(* Logix 5000 project; controller Safety vendor 1 type 14 code 148 rev 32.11; software revision 32.03; part 11 of 17 *)
(* tags used below, declared in another part *)
   ExBridle_DrvsOff : BOOL;   // Exit Bridle Drives OFF ( 1= OFF)
   ExBridle_SafeOffEn : BOOL;   // Exit Bridle Safe-Off Enable ( 1= Enable )
   ExBridle_SafeOffFltRst : BOOL;   // Exit Bridle Safe-Off Fault Reset ( 1= Reset Cmd )
   Line_TotalMode : BOOL;   // Line TOTAL Mode ( 1= Total Mode) (0 = Coil to Coil)
   LineSts : UDT_SysStatus;
   PW_DrvsOff : BOOL;   // Paper Winder Drives OFF ( 1= OFF)
   PW_SafeTrqEn : BOOL;   // Paper Winder Safe-Trq Off Enable ( 1= Enable )
   Rew_DrvsOff : BOOL;   // Rewind Drives OFF ( 1= OFF)
   REW_SafeOffEn : BOOL;   // Rewind Safe-Off Enable ( 1= Enable )
   REW_SafeOffFltRst : BOOL;   // Rewind Safe-Off Fault Reset ( 1= Reset Cmd )
   SafeOff_y172CR460 : CONFIGURABLE_ROUT;   // Shear Die Main Contactor Relay
   SafeOff_y172CR460_Flt : ALIAS FOR Flt_SafeOff[0].0;   // Shear Die Main Contactor Relay Fault ( 1= Fault)
   SafeOff_y172CR510 : CONFIGURABLE_ROUT;   // Shear Die Drive Enable Relay
   SafeOff_y172CR510_Flt : ALIAS FOR Flt_SafeOff[0].1;   // Shear Die Drive Enable Relay Fault ( 1= Fault)
   SafeOff_y614CR040 : CONFIGURABLE_ROUT;   // #1 Exit Bridle Roll 6 Main Contactor Relay
   SafeOff_y614CR040_Flt : ALIAS FOR Flt_SafeOff[0].10;   // #1 Exit Bridle Roll 6 Main Contactor Relay Fault ( 1= Fault)
   SafeOff_y614CR090 : CONFIGURABLE_ROUT;   // #1 Exit Bridle Roll 6 Drive Enable Relay
   SafeOff_y614CR090_Flt : ALIAS FOR Flt_SafeOff[0].11;   // #1 Exit Bridle Roll 6 Drive Enable Relay Fault ( 1= Fault)
   SafeOff_y614CR130 : CONFIGURABLE_ROUT;   // #2 Exit Bridle Roll 7 Main Contactor Relay
   SafeOff_y614CR130_Flt : ALIAS FOR Flt_SafeOff[0].12;   // #2 Exit Bridle Roll 7 Main Contactor Relay Fault ( 1= Fault)
   SafeOff_y614CR170 : CONFIGURABLE_ROUT;   // #2 Exit Bridle Roll 7 Drive Enable Relay
   SafeOff_y614CR170_Flt : ALIAS FOR Flt_SafeOff[0].13;   // #2 Exit Bridle Roll 7 Drive Enable Relay Fault ( 1= Fault)
   SafeOff_y614CR210 : CONFIGURABLE_ROUT;   // Rewind Main Contactor Relay
   SafeOff_y614CR210_Flt : ALIAS FOR Flt_SafeOff[0].14;   // Rewind Main Contactor Relay Fault ( 1= Fault)
   SafeOff_y614CR250 : CONFIGURABLE_ROUT;   // Rewind Drive Enable Relay
   SafeOff_y614CR250_Flt : ALIAS FOR Flt_SafeOff[0].15;   // Rewind Drive Enable Relay Fault ( 1= Fault)
   SC_DrvsOff : BOOL;   // Scrap Chop Conveyor Drives OFF ( 1= OFF)
   SC_SafeTrqEn : BOOL;   // Scrap Chopper Safe-Trq Off Enable ( 1= Enable )
   SGWA_DrvsOff : BOOL;   // Side Guide Width Adjust Drives OFF ( 1= OFF)
   SGWA_SafeTrqEn : BOOL;   // Side Guide Width Adjust Safe-Trq Off Enable ( 1= Enable )
   ShearSts : UDT_ShearStatus;
   SrDie_DrvsOff : BOOL;   // Shear Die Drives OFF ( 1= OFF)
   SrDie_SafeOffEn : BOOL;   // Shear Die Safe-Off Enable ( 1= Enable )
   SrDie_SafeOffFltRst : BOOL;   // Shear Die Safe-Off Fault Reset ( 1= Reset Cmd )
   TK_DrvsOff : BOOL;   // Trimmer Knives/ Width Adjust Drives OFF ( 1= OFF)
   TK_SafeTrqEn : BOOL;   // Trimmer Knife Safe-Trq Off Enable ( 1= Enable )
   UnPR_DrvsOff : BOOL;   // Unwind Pinch Roll Drives OFF ( 1= OFF)
   UnPR_SafeTrqEn : BOOL;   // Unwind Pinch Roll Safe-Trq Off Enable ( 1= Enable )
   WTPR_DrvsOff : BOOL;   // Wash Tank Pinch Rolls (1-4) Drives OFF ( 1= OFF)
   WTPR_SafeTrqEn : BOOL;   // Wash Tank Pinch Rolls (1-4) Safe-Trq Off Enable ( 1= Enable )
   x172CR460 : ALIAS FOR SDPLC:1:I.Pt00Data;   // Shear Die Drive Main Contactor Safety Relay Input
   x172CR510 : ALIAS FOR SDPLC:1:I.Pt01Data;   // Shear Die Drive Enable Safety Relay Input
   x614CR040 : ALIAS FOR CHPLC:2:I.Pt00Data;   // #1 Exit Bridle Roll 6 Main Contactor Safety Relay
   x614CR090 : ALIAS FOR CHPLC:2:I.Pt01Data;   // #1 Exit Bridle Roll 6 Drive Enable Safety Relay
   x614CR130 : ALIAS FOR CHPLC:2:I.Pt02Data;   // #2 Exit Bridle Roll 7 Main Contactor Safety Relay
   x614CR170 : ALIAS FOR CHPLC:2:I.Pt03Data;   // #2 Exit Bridle Roll 7 Drive Enable Safety Relay
   x614CR210 : ALIAS FOR CHPLC:2:I.Pt04Data;   // Rewind Main Contactor Safety Relay
   x614CR250 : ALIAS FOR CHPLC:2:I.Pt05Data;   // Rewind Drive Enable Safety Relay
   x759MTR080SE : ALIAS FOR MCC3:4:O.Pt02Data;   // Scrap Choppers Width Adjust Safety Enable
   x759MTR080SP : ALIAS FOR MCC3:4:O.Pt01Data;   // Scrap Choppers Width Adjust Safety Power
   y172CR460 : ALIAS FOR SDPLC:2:O.Pt00Data;   // Shear Die Drive Main Contactor Safety Relay Output
   y172CR510 : ALIAS FOR SDPLC:2:O.Pt01Data;   // Shear Die Drive Enable Safety Relay Output
   y614CR040 : ALIAS FOR CHPLC:5:O.Pt00Data;   // #1 Exit Bridle Roll 6 Main Contactor Safety Relay
   y614CR090 : ALIAS FOR CHPLC:5:O.Pt01Data;   // #1 Exit Bridle Roll 6 Drive Enable Safety Relay
   y614CR130 : ALIAS FOR CHPLC:5:O.Pt02Data;   // #2 Exit Bridle Roll 7 Main Contactor Safety Relay
   y614CR170 : ALIAS FOR CHPLC:5:O.Pt03Data;   // #2 Exit Bridle Roll 7 Drive Enable Safety Relay
   y614CR210 : ALIAS FOR CHPLC:5:O.Pt04Data;   // Rewind Main Contactor Safety Relay
   y614CR250 : ALIAS FOR CHPLC:5:O.Pt05Data;   // Rewind Drive Enable Safety Relay
   y725MTR080SE : ALIAS FOR MCC2:1:O.Pt01Data;   // Unwind Pinch Roll Safety Enable
   y725MTR080SP : ALIAS FOR MCC2:1:O.Pt00Data;   // Unwind Pinch Roll Safety Power
   y727MTR080SE : ALIAS FOR MCC2:1:O.Pt05Data;   // Paper Winder Safety Enable
   y727MTR080SP : ALIAS FOR MCC2:1:O.Pt04Data;   // Paper Winder Safety Power
   y729MTR080SE : ALIAS FOR MCC2:1:O.Pt03Data;   // Washtank Pinch Roll 4 Safety Enable
   y729MTR080SP : ALIAS FOR MCC2:1:O.Pt02Data;   // Washtank Pinch Roll 4 Safety Power
   y731MTR080SE : ALIAS FOR MCC2:1:O.Pt07Data;   // Washtank Pinch Roll 1 Safety Enable
   y731MTR080SP : ALIAS FOR MCC2:1:O.Pt06Data;   // Washtank Pinch Roll 1 Safety Power
   y733MTR080SE : ALIAS FOR MCC2:2:O.Pt01Data;   // Washtank Pinch Roll 2 Safety Enable
   y733MTR080SP : ALIAS FOR MCC2:2:O.Pt00Data;   // Washtank Pinch Roll 2 Safety Power
   y735MTR080SE : ALIAS FOR MCC2:2:O.Pt03Data;   // Washtank Pinch Roll 3 Safety Enable
   y735MTR080SP : ALIAS FOR MCC2:2:O.Pt02Data;   // Washtank Pinch Roll 3 Safety Power
   y751MTR080SE : ALIAS FOR MCC3:3:O.Pt04Data;   // Trimmer Knives Safety Enable
   y751MTR080SP : ALIAS FOR MCC3:3:O.Pt03Data;   // Trimmer Knives Safety Power
   y754MTR080SE : ALIAS FOR MCC3:3:O.Pt06Data;   // Side Guide Width Adjust Safety Enable
   y754MTR080SP : ALIAS FOR MCC3:3:O.Pt05Data;   // Side Guide Width Adjust Safety Power
   y755MTR080SE : ALIAS FOR MCC3:4:O.Pt00Data;   // Trimmer Knives Width Adjust Safety Enable
   y755MTR080SP : ALIAS FOR MCC3:3:O.Pt07Data;   // Trimmer Knives Width Adjust Safety Power
   y762MTR080SE : ALIAS FOR MCC3:4:O.Pt04Data;   // Scrap Choppers Safety Enable
   y762MTR080SP : ALIAS FOR MCC3:4:O.Pt03Data;   // Scrap Choppers Safety Power
(* SafeOff, continued *)

ROUTINE A03_ExitBridle_CR   (* ladder *)
// Exit Bridle
// Main Contactor and Drive Enable
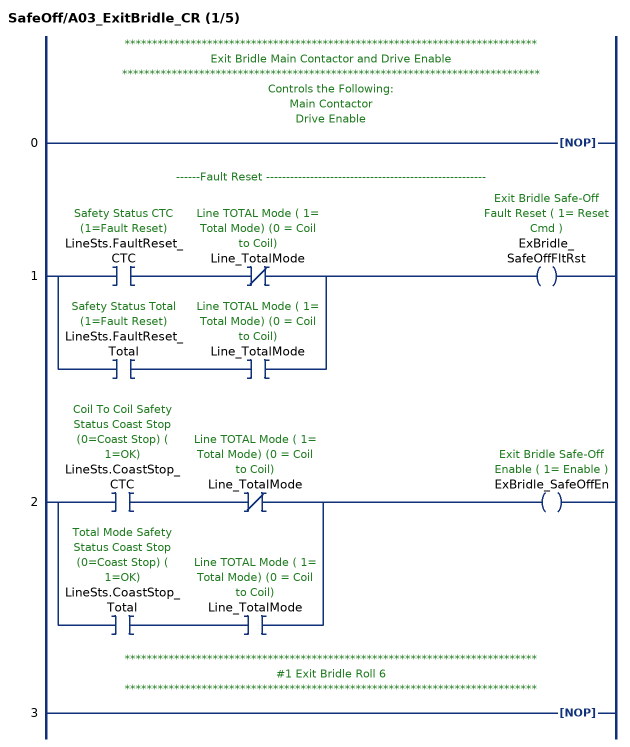
   // ***************************************************************************
   // Exit Bridle Main Contactor and Drive Enable
   // ****************************************************************************
   // Controls the Following:
   // Main Contactor
   // Drive Enable
   0: NOP();
   // ------Fault Reset -------------------------------------------------------
   1: [XIC(LineSts.FaultReset_CTC) XIO(Line_TotalMode) ,XIC(LineSts.FaultReset_Total) XIC(Line_TotalMode) ]OTE(ExBridle_SafeOffFltRst);
   2: [XIC(LineSts.CoastStop_CTC) XIO(Line_TotalMode) ,XIC(LineSts.CoastStop_Total) XIC(Line_TotalMode) ]OTE(ExBridle_SafeOffEn);
   // ***************************************************************************
   // #1 Exit Bridle Roll 6
   // ***************************************************************************
   3: NOP();
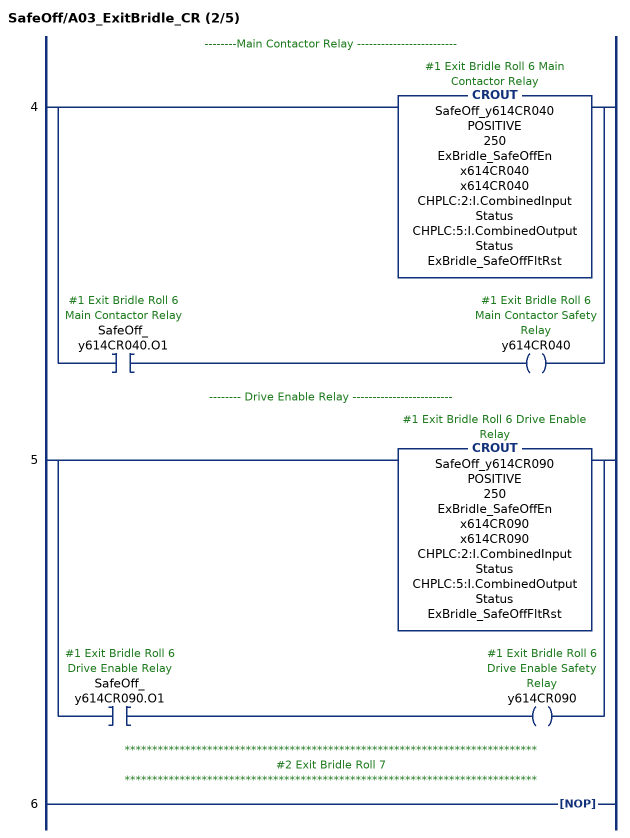
   // --------Main Contactor Relay -------------------------
   4: [CROUT(SafeOff_y614CR040,POSITIVE,250,ExBridle_SafeOffEn,x614CR040,x614CR040,CHPLC:2:I.CombinedInputStatus,CHPLC:5:I.CombinedOutputStatus,ExBridle_SafeOffFltRst) ,XIC(SafeOff_y614CR040.O1) OTE(y614CR040) ];
   // -------- Drive Enable Relay -------------------------
   5: [CROUT(SafeOff_y614CR090,POSITIVE,250,ExBridle_SafeOffEn,x614CR090,x614CR090,CHPLC:2:I.CombinedInputStatus,CHPLC:5:I.CombinedOutputStatus,ExBridle_SafeOffFltRst) ,XIC(SafeOff_y614CR090.O1) OTE(y614CR090) ];
   // ***************************************************************************
   // #2 Exit Bridle Roll 7
   // ***************************************************************************
   6: NOP();
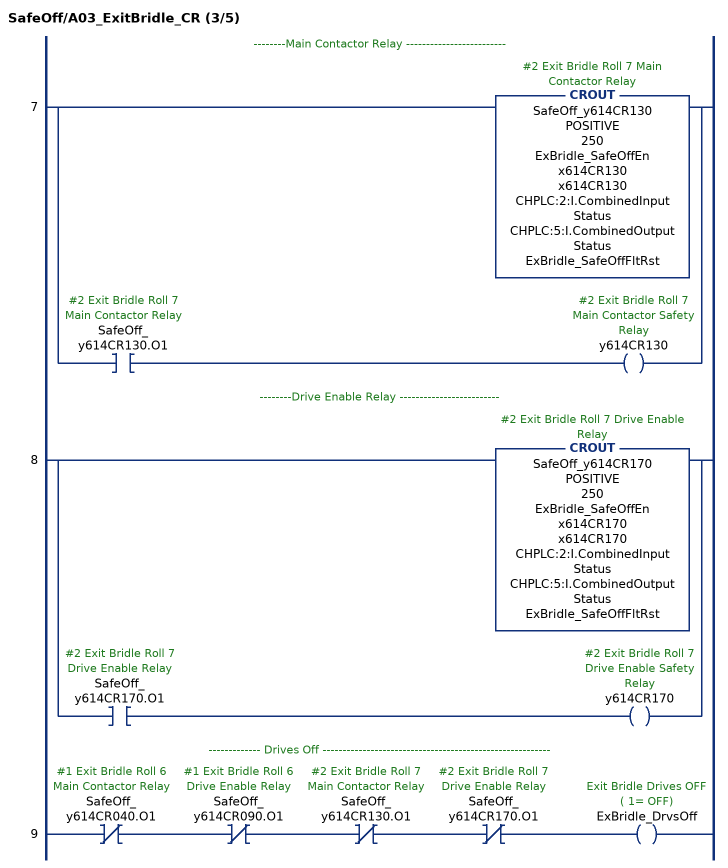
   // --------Main Contactor Relay -------------------------
   7: [CROUT(SafeOff_y614CR130,POSITIVE,250,ExBridle_SafeOffEn,x614CR130,x614CR130,CHPLC:2:I.CombinedInputStatus,CHPLC:5:I.CombinedOutputStatus,ExBridle_SafeOffFltRst) ,XIC(SafeOff_y614CR130.O1) OTE(y614CR130) ];
   // --------Drive Enable Relay -------------------------
   8: [CROUT(SafeOff_y614CR170,POSITIVE,250,ExBridle_SafeOffEn,x614CR170,x614CR170,CHPLC:2:I.CombinedInputStatus,CHPLC:5:I.CombinedOutputStatus,ExBridle_SafeOffFltRst) ,XIC(SafeOff_y614CR170.O1) OTE(y614CR170) ];
   // ------------- Drives Off ---------------------------------------------------------
   9: XIO(SafeOff_y614CR040.O1)XIO(SafeOff_y614CR090.O1)XIO(SafeOff_y614CR130.O1)XIO(SafeOff_y614CR170.O1)OTE(ExBridle_DrvsOff);
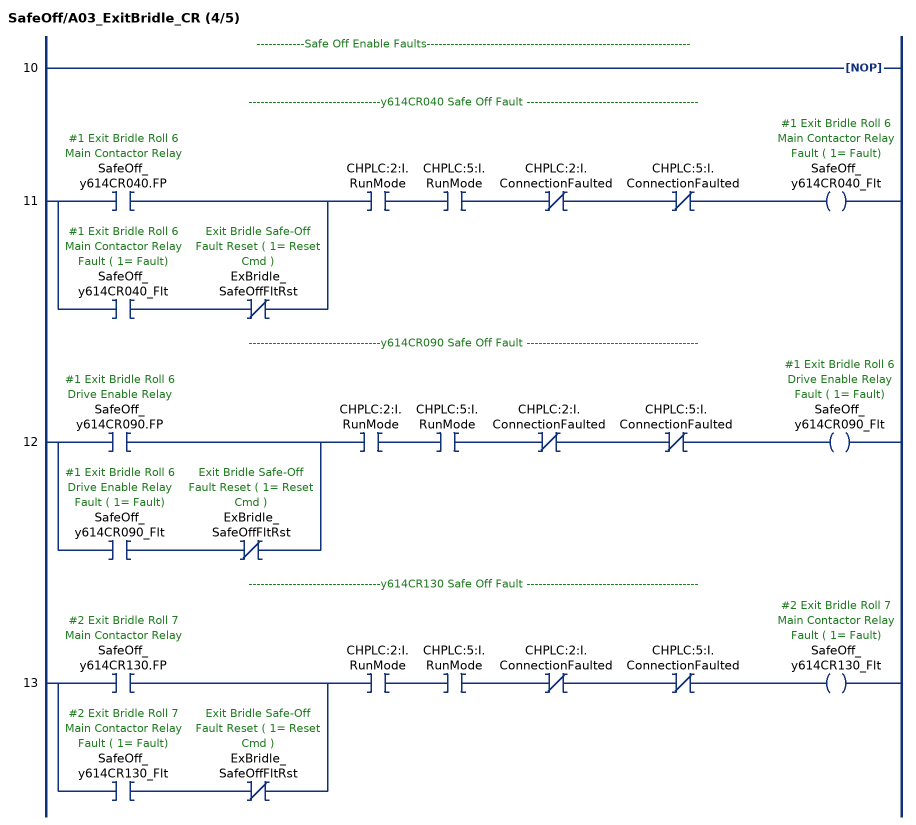
   // ------------Safe Off Enable Faults------------------------------------------------------------------
   10: NOP();
   // ---------------------------------y614CR040 Safe Off Fault -------------------------------------------
   11: [XIC(SafeOff_y614CR040.FP) ,XIC(SafeOff_y614CR040_Flt) XIO(ExBridle_SafeOffFltRst) ]XIC(CHPLC:2:I.RunMode)XIC(CHPLC:5:I.RunMode)XIO(CHPLC:2:I.ConnectionFaulted)XIO(CHPLC:5:I.ConnectionFaulted)OTE(SafeOff_y614CR040_Flt);
   // ---------------------------------y614CR090 Safe Off Fault -------------------------------------------
   12: [XIC(SafeOff_y614CR090.FP) ,XIC(SafeOff_y614CR090_Flt) XIO(ExBridle_SafeOffFltRst) ]XIC(CHPLC:2:I.RunMode)XIC(CHPLC:5:I.RunMode)XIO(CHPLC:2:I.ConnectionFaulted)XIO(CHPLC:5:I.ConnectionFaulted)OTE(SafeOff_y614CR090_Flt);
   // ---------------------------------y614CR130 Safe Off Fault -------------------------------------------
   13: [XIC(SafeOff_y614CR130.FP) ,XIC(SafeOff_y614CR130_Flt) XIO(ExBridle_SafeOffFltRst) ]XIC(CHPLC:2:I.RunMode)XIC(CHPLC:5:I.RunMode)XIO(CHPLC:2:I.ConnectionFaulted)XIO(CHPLC:5:I.ConnectionFaulted)OTE(SafeOff_y614CR130_Flt);
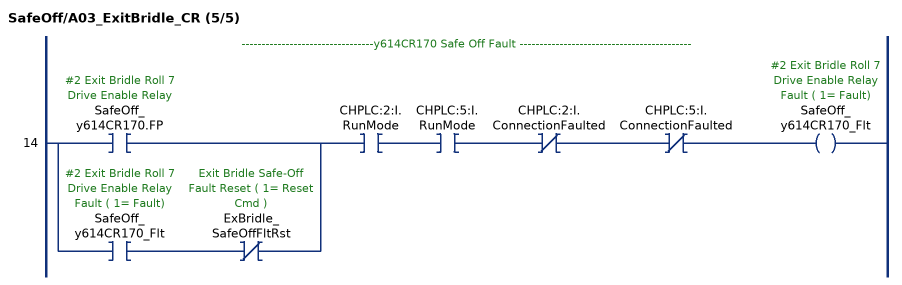
   // ---------------------------------y614CR170 Safe Off Fault -------------------------------------------
   14: [XIC(SafeOff_y614CR170.FP) ,XIC(SafeOff_y614CR170_Flt) XIO(ExBridle_SafeOffFltRst) ]XIC(CHPLC:2:I.RunMode)XIC(CHPLC:5:I.RunMode)XIO(CHPLC:2:I.ConnectionFaulted)XIO(CHPLC:5:I.ConnectionFaulted)OTE(SafeOff_y614CR170_Flt);
END_ROUTINE

ROUTINE A04_Rewind_CR   (* ladder *)
// Rewind
// Main Contactor and Drive Enable
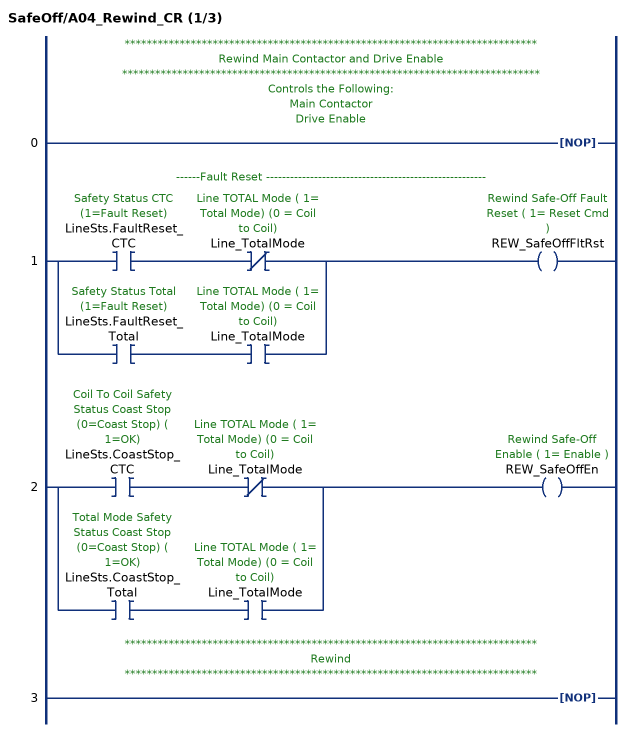
   // ***************************************************************************
   // Rewind Main Contactor and Drive Enable
   // ****************************************************************************
   // Controls the Following:
   // Main Contactor
   // Drive Enable
   0: NOP();
   // ------Fault Reset -------------------------------------------------------
   1: [XIC(LineSts.FaultReset_CTC) XIO(Line_TotalMode) ,XIC(LineSts.FaultReset_Total) XIC(Line_TotalMode) ]OTE(REW_SafeOffFltRst);
   2: [XIC(LineSts.CoastStop_CTC) XIO(Line_TotalMode) ,XIC(LineSts.CoastStop_Total) XIC(Line_TotalMode) ]OTE(REW_SafeOffEn);
   // ***************************************************************************
   // Rewind
   // ***************************************************************************
   3: NOP();
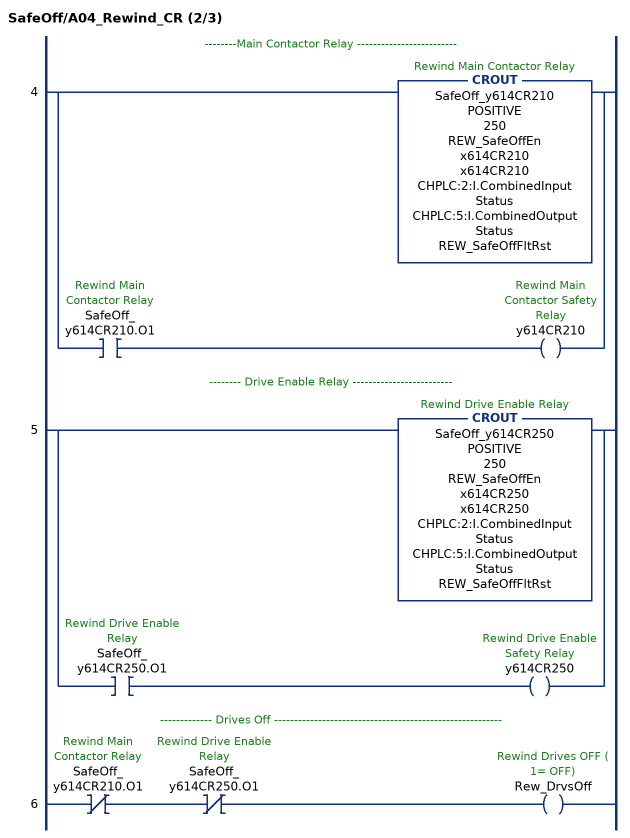
   // --------Main Contactor Relay -------------------------
   4: [CROUT(SafeOff_y614CR210,POSITIVE,250,REW_SafeOffEn,x614CR210,x614CR210,CHPLC:2:I.CombinedInputStatus,CHPLC:5:I.CombinedOutputStatus,REW_SafeOffFltRst) ,XIC(SafeOff_y614CR210.O1) OTE(y614CR210) ];
   // -------- Drive Enable Relay -------------------------
   5: [CROUT(SafeOff_y614CR250,POSITIVE,250,REW_SafeOffEn,x614CR250,x614CR250,CHPLC:2:I.CombinedInputStatus,CHPLC:5:I.CombinedOutputStatus,REW_SafeOffFltRst) ,XIC(SafeOff_y614CR250.O1) OTE(y614CR250) ];
   // ------------- Drives Off ---------------------------------------------------------
   6: XIO(SafeOff_y614CR210.O1)XIO(SafeOff_y614CR250.O1)OTE(Rew_DrvsOff);
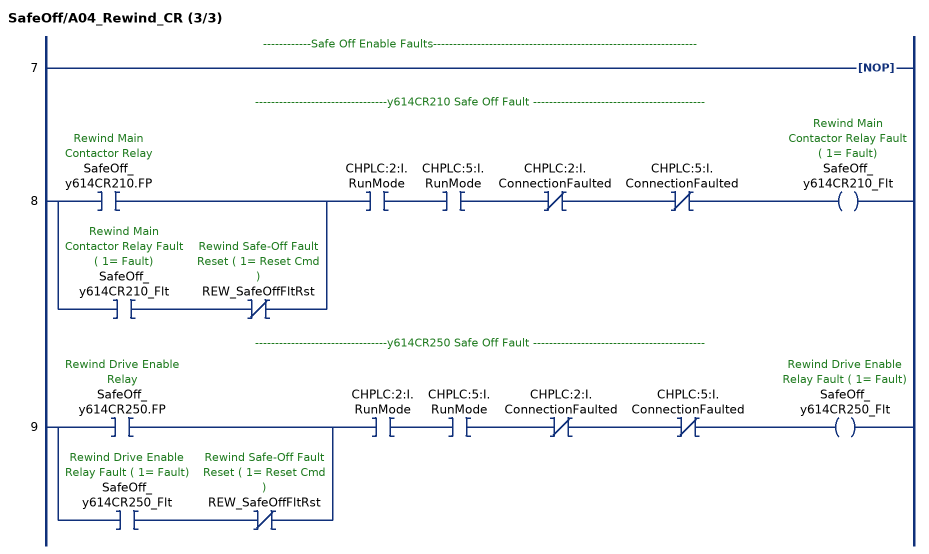
   // ------------Safe Off Enable Faults------------------------------------------------------------------
   7: NOP();
   // ---------------------------------y614CR210 Safe Off Fault -------------------------------------------
   8: [XIC(SafeOff_y614CR210.FP) ,XIC(SafeOff_y614CR210_Flt) XIO(REW_SafeOffFltRst) ]XIC(CHPLC:2:I.RunMode)XIC(CHPLC:5:I.RunMode)XIO(CHPLC:2:I.ConnectionFaulted)XIO(CHPLC:5:I.ConnectionFaulted)OTE(SafeOff_y614CR210_Flt);
   // ---------------------------------y614CR250 Safe Off Fault -------------------------------------------
   9: [XIC(SafeOff_y614CR250.FP) ,XIC(SafeOff_y614CR250_Flt) XIO(REW_SafeOffFltRst) ]XIC(CHPLC:2:I.RunMode)XIC(CHPLC:5:I.RunMode)XIO(CHPLC:2:I.ConnectionFaulted)XIO(CHPLC:5:I.ConnectionFaulted)OTE(SafeOff_y614CR250_Flt);
END_ROUTINE

ROUTINE A05_ShearDie_CR   (* ladder *)
// Shear Die Accelerator
// Main Contactor and Drive Enable
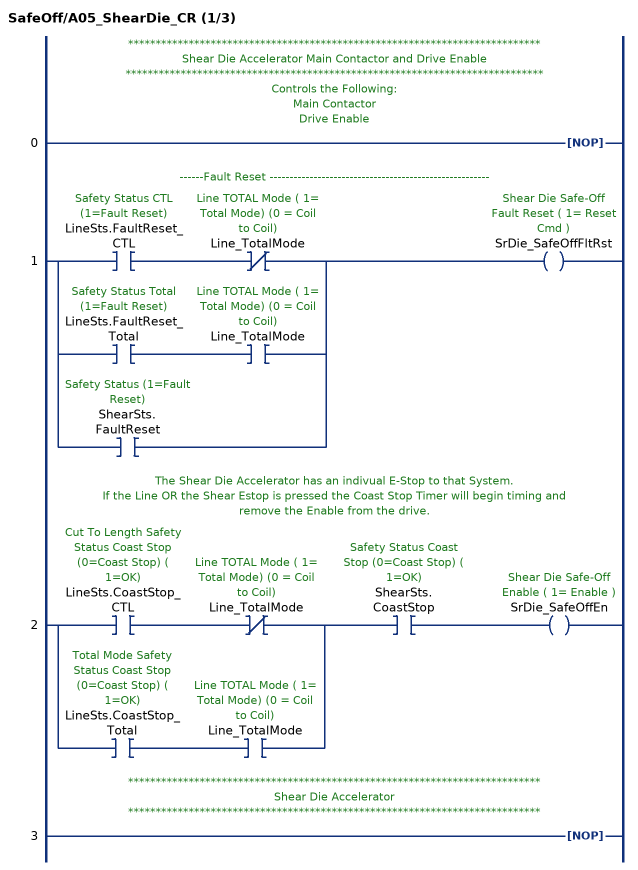
   // ***************************************************************************
   // Shear Die Accelerator Main Contactor and Drive Enable
   // ****************************************************************************
   // Controls the Following:
   // Main Contactor
   // Drive Enable
   0: NOP();
   // ------Fault Reset -------------------------------------------------------
   1: [XIC(LineSts.FaultReset_CTL) XIO(Line_TotalMode) ,XIC(LineSts.FaultReset_Total) XIC(Line_TotalMode) ,XIC(ShearSts.FaultReset) ]OTE(SrDie_SafeOffFltRst);
   // The Shear Die Accelerator has an indivual E-Stop to that System.
   // If the Line OR the Shear Estop is pressed the Coast Stop Timer will begin timing and
   // remove the Enable from the drive.
   2: [XIC(LineSts.CoastStop_CTL) XIO(Line_TotalMode) ,XIC(LineSts.CoastStop_Total) XIC(Line_TotalMode) ]XIC(ShearSts.CoastStop)OTE(SrDie_SafeOffEn);
   // ***************************************************************************
   // Shear Die Accelerator
   // ***************************************************************************
   3: NOP();
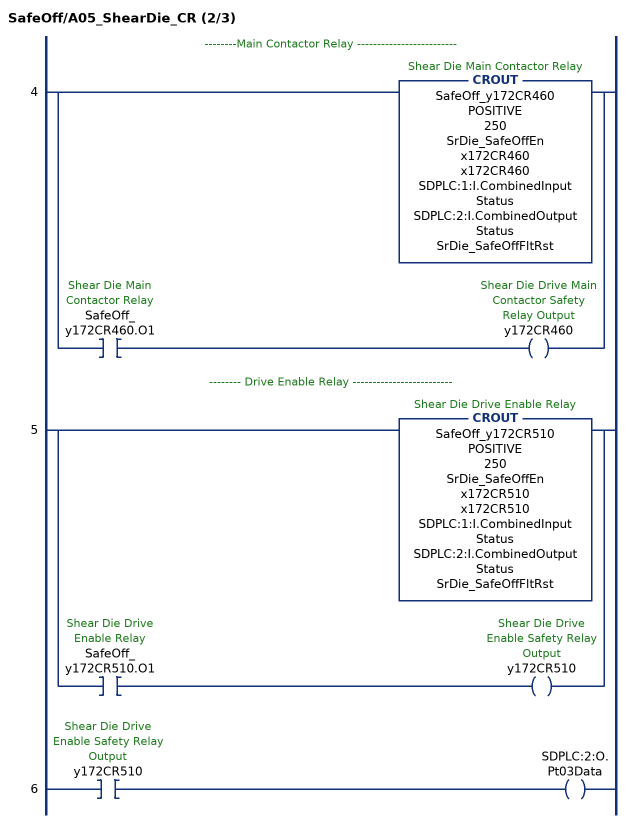
   // --------Main Contactor Relay -------------------------
   4: [CROUT(SafeOff_y172CR460,POSITIVE,250,SrDie_SafeOffEn,x172CR460,x172CR460,SDPLC:1:I.CombinedInputStatus,SDPLC:2:I.CombinedOutputStatus,SrDie_SafeOffFltRst) ,XIC(SafeOff_y172CR460.O1) OTE(y172CR460) ];
   // -------- Drive Enable Relay -------------------------
   5: [CROUT(SafeOff_y172CR510,POSITIVE,250,SrDie_SafeOffEn,x172CR510,x172CR510,SDPLC:1:I.CombinedInputStatus,SDPLC:2:I.CombinedOutputStatus,SrDie_SafeOffFltRst) ,XIC(SafeOff_y172CR510.O1) OTE(y172CR510) ];
   6: XIC(y172CR510)OTE(SDPLC:2:O.Pt03Data);
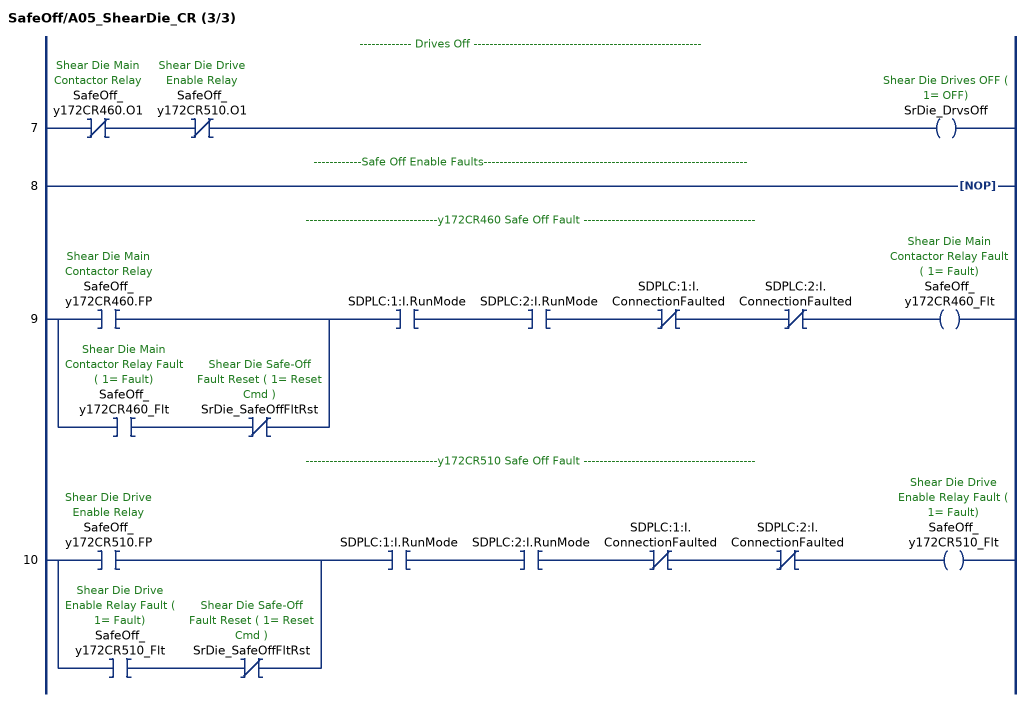
   // ------------- Drives Off ---------------------------------------------------------
   7: XIO(SafeOff_y172CR460.O1)XIO(SafeOff_y172CR510.O1)OTE(SrDie_DrvsOff);
   // ------------Safe Off Enable Faults------------------------------------------------------------------
   8: NOP();
   // ---------------------------------y172CR460 Safe Off Fault -------------------------------------------
   9: [XIC(SafeOff_y172CR460.FP) ,XIC(SafeOff_y172CR460_Flt) XIO(SrDie_SafeOffFltRst) ]XIC(SDPLC:1:I.RunMode)XIC(SDPLC:2:I.RunMode)XIO(SDPLC:1:I.ConnectionFaulted)XIO(SDPLC:2:I.ConnectionFaulted)OTE(SafeOff_y172CR460_Flt);
   // ---------------------------------y172CR510 Safe Off Fault -------------------------------------------
   10: [XIC(SafeOff_y172CR510.FP) ,XIC(SafeOff_y172CR510_Flt) XIO(SrDie_SafeOffFltRst) ]XIC(SDPLC:1:I.RunMode)XIC(SDPLC:2:I.RunMode)XIO(SDPLC:1:I.ConnectionFaulted)XIO(SDPLC:2:I.ConnectionFaulted)OTE(SafeOff_y172CR510_Flt);
END_ROUTINE

ROUTINE B01_UnPR_SafeTrqOff   (* ladder *)
// Unwind Pinch Roll
// Safety Power Enable
// (Safe Trq Off and Drv Enable)
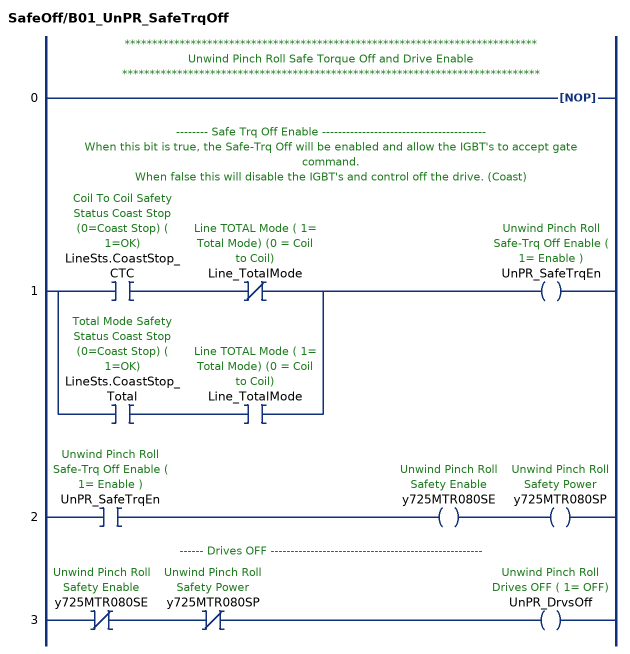
   // ***************************************************************************
   // Unwind Pinch Roll Safe Torque Off and Drive Enable
   // ****************************************************************************
   0: NOP();
   // -------- Safe Trq Off Enable -----------------------------------------
   // When this bit is true, the Safe-Trq Off will be enabled and allow the IGBT's to accept gate command.
   // When false this will disable the IGBT's and control off the drive. (Coast)
   1: [XIC(LineSts.CoastStop_CTC) XIO(Line_TotalMode) ,XIC(LineSts.CoastStop_Total) XIC(Line_TotalMode) ]OTE(UnPR_SafeTrqEn);
   2: XIC(UnPR_SafeTrqEn)OTE(y725MTR080SE)OTE(y725MTR080SP);
   // ------ Drives OFF -----------------------------------------------------
   3: XIO(y725MTR080SE)XIO(y725MTR080SP)OTE(UnPR_DrvsOff);
END_ROUTINE

ROUTINE B02_PW_SafeTrqOff   (* ladder *)
// Paper Winder
// Safety Power Enable
// (Safe Trq Off and Drv Enable)
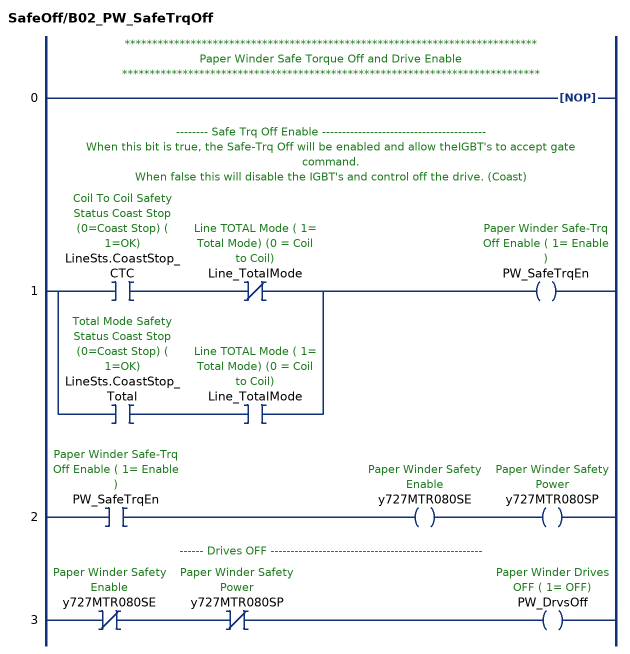
   // ***************************************************************************
   // Paper Winder Safe Torque Off and Drive Enable
   // ****************************************************************************
   0: NOP();
   // -------- Safe Trq Off Enable -----------------------------------------
   // When this bit is true, the Safe-Trq Off will be enabled and allow theIGBT's to accept gate command.
   // When false this will disable the IGBT's and control off the drive. (Coast)
   1: [XIC(LineSts.CoastStop_CTC) XIO(Line_TotalMode) ,XIC(LineSts.CoastStop_Total) XIC(Line_TotalMode) ]OTE(PW_SafeTrqEn);
   2: XIC(PW_SafeTrqEn)OTE(y727MTR080SE)OTE(y727MTR080SP);
   // ------ Drives OFF -----------------------------------------------------
   3: XIO(y727MTR080SE)XIO(y727MTR080SP)OTE(PW_DrvsOff);
END_ROUTINE

ROUTINE B03_TK_SafeTrqOff   (* ladder *)
// Trimmer Knife, Width Adjust
// Safety Power Enable
// (Safe Trq Off and Drv Enable)
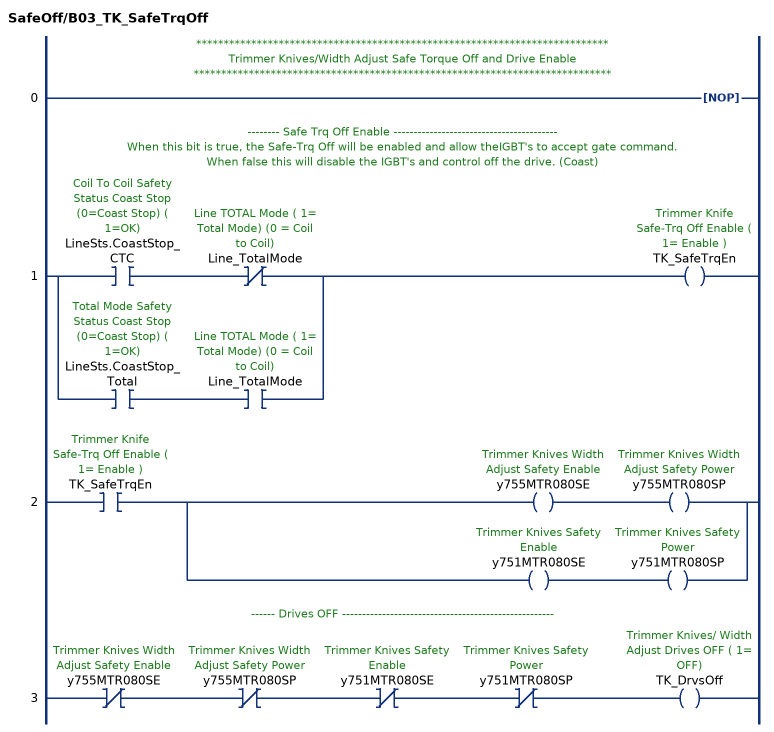
   // ***************************************************************************
   // Trimmer Knives/Width Adjust Safe Torque Off and Drive Enable
   // ****************************************************************************
   0: NOP();
   // -------- Safe Trq Off Enable -----------------------------------------
   // When this bit is true, the Safe-Trq Off will be enabled and allow theIGBT's to accept gate command.
   // When false this will disable the IGBT's and control off the drive. (Coast)
   1: [XIC(LineSts.CoastStop_CTC) XIO(Line_TotalMode) ,XIC(LineSts.CoastStop_Total) XIC(Line_TotalMode) ]OTE(TK_SafeTrqEn);
   2: XIC(TK_SafeTrqEn)[OTE(y755MTR080SE) OTE(y755MTR080SP) ,OTE(y751MTR080SE) OTE(y751MTR080SP) ];
   // ------ Drives OFF -----------------------------------------------------
   3: XIO(y755MTR080SE)XIO(y755MTR080SP)XIO(y751MTR080SE)XIO(y751MTR080SP)OTE(TK_DrvsOff);
END_ROUTINE

ROUTINE B04_SC_SafeTrqOff   (* ladder *)
// Scrap Chopper
// Safety Power Enable
// (Safe Trq Off and Drv Enable)
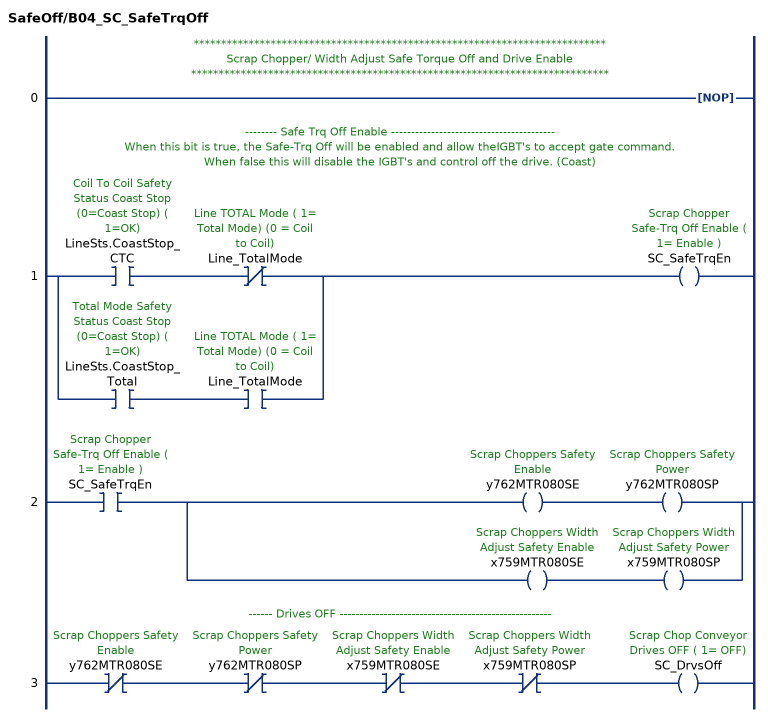
   // ***************************************************************************
   // Scrap Chopper/ Width Adjust Safe Torque Off and Drive Enable
   // ****************************************************************************
   0: NOP();
   // -------- Safe Trq Off Enable -----------------------------------------
   // When this bit is true, the Safe-Trq Off will be enabled and allow theIGBT's to accept gate command.
   // When false this will disable the IGBT's and control off the drive. (Coast)
   1: [XIC(LineSts.CoastStop_CTC) XIO(Line_TotalMode) ,XIC(LineSts.CoastStop_Total) XIC(Line_TotalMode) ]OTE(SC_SafeTrqEn);
   2: XIC(SC_SafeTrqEn)[OTE(y762MTR080SE) OTE(y762MTR080SP) ,OTE(x759MTR080SE) OTE(x759MTR080SP) ];
   // ------ Drives OFF -----------------------------------------------------
   3: XIO(y762MTR080SE)XIO(y762MTR080SP)XIO(x759MTR080SE)XIO(x759MTR080SP)OTE(SC_DrvsOff);
END_ROUTINE

ROUTINE B05_WTPR_SafeTrqOff   (* ladder *)
// Wash Tank Pinch Rolls
// Safety Power Enable
// (Safe Trq Off and Drv Enable)
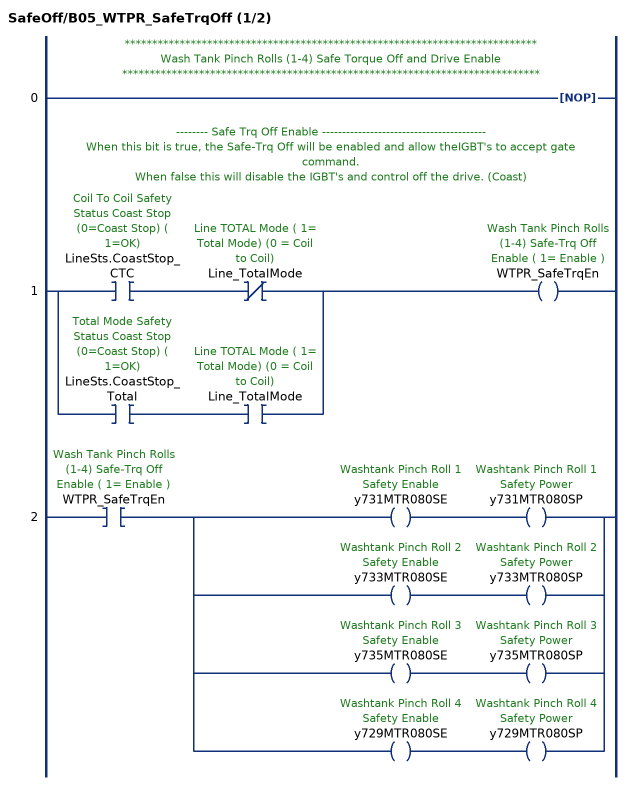
   // ***************************************************************************
   // Wash Tank Pinch Rolls (1-4) Safe Torque Off and Drive Enable
   // ****************************************************************************
   0: NOP();
   // -------- Safe Trq Off Enable -----------------------------------------
   // When this bit is true, the Safe-Trq Off will be enabled and allow theIGBT's to accept gate command.
   // When false this will disable the IGBT's and control off the drive. (Coast)
   1: [XIC(LineSts.CoastStop_CTC) XIO(Line_TotalMode) ,XIC(LineSts.CoastStop_Total) XIC(Line_TotalMode) ]OTE(WTPR_SafeTrqEn);
   2: XIC(WTPR_SafeTrqEn)[OTE(y731MTR080SE) OTE(y731MTR080SP) ,OTE(y733MTR080SE) OTE(y733MTR080SP) ,OTE(y735MTR080SE) OTE(y735MTR080SP) ,OTE(y729MTR080SE) OTE(y729MTR080SP) ];
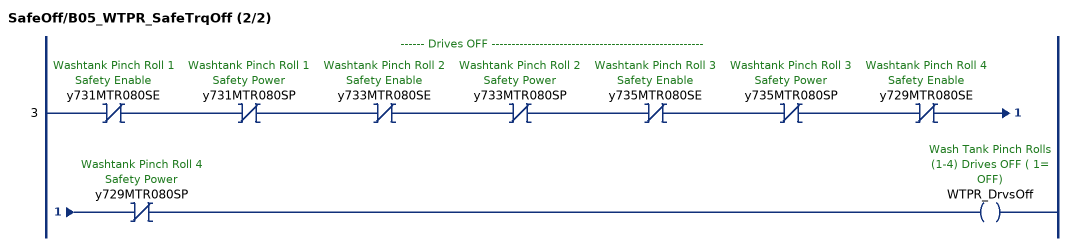
   // ------ Drives OFF -----------------------------------------------------
   3: XIO(y731MTR080SE)XIO(y731MTR080SP)XIO(y733MTR080SE)XIO(y733MTR080SP)XIO(y735MTR080SE)XIO(y735MTR080SP)XIO(y729MTR080SE)XIO(y729MTR080SP)OTE(WTPR_DrvsOff);
END_ROUTINE

ROUTINE B06_SGWA_SafeTrqOff   (* ladder *)
// Side Guide Width Adjust
// Safety Power Enable
// (Safe Trq Off and Drv Enable)
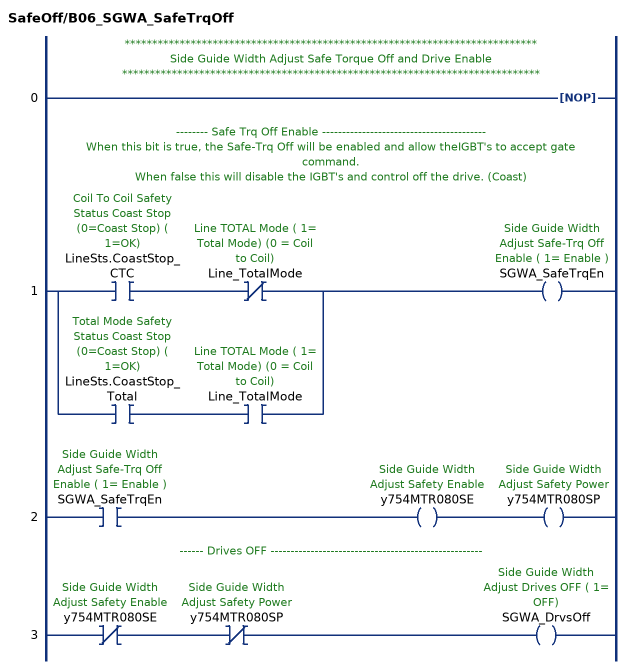
   // ***************************************************************************
   // Side Guide Width Adjust Safe Torque Off and Drive Enable
   // ****************************************************************************
   0: NOP();
   // -------- Safe Trq Off Enable -----------------------------------------
   // When this bit is true, the Safe-Trq Off will be enabled and allow theIGBT's to accept gate command.
   // When false this will disable the IGBT's and control off the drive. (Coast)
   1: [XIC(LineSts.CoastStop_CTC) XIO(Line_TotalMode) ,XIC(LineSts.CoastStop_Total) XIC(Line_TotalMode) ]OTE(SGWA_SafeTrqEn);
   2: XIC(SGWA_SafeTrqEn)OTE(y754MTR080SE)OTE(y754MTR080SP);
   // ------ Drives OFF -----------------------------------------------------
   3: XIO(y754MTR080SE)XIO(y754MTR080SP)OTE(SGWA_DrvsOff);
END_ROUTINE
